INTERFACE iMover

METHOD ActivateTrack : BOOL
VAR_INPUT
	Track	: REFERENCE TO Track;
END_VAR
END_METHOD

{attribute 'monitoring' := 'call'}
PROPERTY CurrentDestinationPosition : LREAL
GET
END_GET
END_PROPERTY

{attribute 'monitoring' := 'call'}
PROPERTY CurrentMoveType : MoverCommandType_enum
GET
END_GET
END_PROPERTY

PROPERTY CurrentObjective : String
GET
END_GET
END_PROPERTY

PROPERTY CurrentTrack : POINTER TO Track
GET
END_GET
END_PROPERTY

METHOD Cyclic : iMover
VAR_IN_OUT
	GroupReference		: AXES_GROUP_REF;
END_VAR
END_METHOD

METHOD CyclicTrack : BOOL
VAR
END_VAR
END_METHOD

METHOD Disable : iMover
VAR_INPUT
END_VAR
END_METHOD

METHOD Enable : iMover
VAR_INPUT
END_VAR
END_METHOD

METHOD GroupStop : iMover
VAR_INPUT
END_VAR
END_METHOD

METHOD Halt : iMover
VAR_INPUT
END_VAR
END_METHOD

PROPERTY IsTrackReady : BOOL
GET
END_GET
END_PROPERTY

METHOD LogUserEvent : iMover
VAR_INPUT
	String1	: STRING;	// First content section of user-event message
	String2 : STRING;	// Second content section of user-event message
	String3 : STRING;	// Third content section of user-event message
END_VAR
END_METHOD

METHOD PUBLIC MoveToPosition : iMover
VAR_INPUT
	
	DestinationPosition		: LREAL;	// position on track for a shuttle to move towards

END_VAR
END_METHOD

METHOD MoveToStation : iMover
VAR_INPUT
	DestinationStation	: REFERENCE TO Station;	
END_VAR
END_METHOD

METHOD MoveVelocity : iMover
VAR_INPUT
	DesiredVelocity : LREAL;		//The velocity to be commanded [mm/s]
END_VAR
END_METHOD

PROPERTY Payload : Payload_TYP
GET
END_GET
SET
END_SET
END_PROPERTY

METHOD ReissueCommand : iMover
VAR_INPUT
END_VAR
END_METHOD


METHOD SetAcceleration : iMover
VAR_INPUT
	Acceleration	: LREAL;
END_VAR
END_METHOD

METHOD SetDeceleration : iMover
VAR_INPUT
	Deceleration	: LREAL;
END_VAR
END_METHOD

METHOD SetDirection : iMover
VAR_INPUT
	Direction		: Tc3_Mc3Definitions.MC_Direction;
END_VAR
END_METHOD

METHOD SetJerk : iMover
VAR_INPUT
	Jerk		: LREAL;
END_VAR
END_METHOD

METHOD SetVelocity : iMover
VAR_INPUT
	Velocity		: LREAL;		// Updates Mover's internal velocity parameter. Takes effect immediately. [mm/s]
END_VAR
END_METHOD

METHOD SyncToAxis : iMover
VAR_INPUT
	
	MasterAxis		: REFERENCE TO AXIS_REF;
	MasterSyncPos	: LREAL;	// Master sync position (nonmodulo), where the input axis will be located when first synchronized
	SlaveSyncPos	: LREAL;	// Mover sync position, where the mover will be located when first synchronized
	SyncStrategy	: MC_SYNC_STRATEGY;	// Direction input
	
END_VAR
END_METHOD

METHOD SyncToMover : iMover
VAR_INPUT

	MasterMover		: REFERENCE TO Mover;	// Synchronization master mover, whose position to follow. Further motion commands break the pairing
	Gap				: LREAL;				// Gap distance to lead mover. Positive values indicate following, negative values indicate leading

END_VAR
END_METHOD

END_INTERFACE

(* stored: Version 1.1.0.1, ProductVersion 3.1.4024.12
   Itf iMover: Id {30ffe45f-c01a-49ae-9d19-23395eddd7e8}
   Folder Methods: Id {1b23c83c-1258-4c4f-a9ad-a029b20875d0}
   Folder Properties: Id {73a4fa43-0d07-4dea-a761-2d7dc373ee4f}
   Method ActivateTrack: Id {0340ebdc-9de8-0f0c-175a-ccd19ec99ec0}
   Property CurrentDestinationPosition: Id {fd336655-1b12-4c85-8800-888e616a0190}
   Get Get: Id {3855cb66-22eb-461a-b098-b3ca2fe0f4f3}
   Property CurrentMoveType: Id {f31956ff-9981-42ba-a963-53182be5a6a1}
   Get Get: Id {4f4d6df0-727b-4d83-aa6a-31cf10efdd21}
   Property CurrentObjective: Id {8ebf7eff-2b0b-45f9-8604-dc48a6c2dec6}
   Get Get: Id {1c8cee4d-d0d3-4396-aef2-3ace7cdfef3e}
   Property CurrentTrack: Id {6df508fb-5bd5-0e4f-32b6-ad8f8b706833}
   Get Get: Id {a9690824-dbea-0ac9-0859-6bf4b97c3449}
   Method Cyclic: Id {b891277c-4d72-4aed-a650-47e395d59c1f}
   Method CyclicTrack: Id {3e3500dc-85cc-0f0e-23f9-0a487fad9df8}
   Method Disable: Id {d596b2ea-b33b-4163-8d7c-887245d1fbda}
   Method Enable: Id {9670332c-ffbe-4d1e-8081-d250b5368f10}
   Method GroupStop: Id {3415d362-731d-4eed-aa29-ec6fe9ada72d}
   Method Halt: Id {75fb2e90-af06-4361-8343-b02ee21a7773}
   Property IsTrackReady: Id {a749704e-a727-05fa-1be8-d11fd5732682}
   Get Get: Id {3d58532e-56d6-0a5a-0811-67af41cc16bc}
   Method LogUserEvent: Id {24391ec1-ea2c-453c-9dee-5da9dcff0b7b}
   Method MoveToPosition: Id {12a28052-bce3-440a-bab1-51b28f359a72}
   Method MoveToStation: Id {1d1440c0-f172-4e49-adaf-b20085e83a8c}
   Method MoveVelocity: Id {86b32a6f-8247-4d7d-b5bb-30abae20d537}
   Property Payload: Id {8debfc3a-ede6-452a-8f81-b4825ce39b3b}
   Get Get: Id {80534c46-bb57-4e05-bca0-e1e88d880aac}
   Set Set: Id {f79463b1-b92f-424b-a739-aa6b1256efa9}
   Method ReissueCommand: Id {1fc1edba-27e0-4034-90b8-62d930acd5b9}
   Method SetAcceleration: Id {8d0e79e2-9192-4e14-ba95-b7dae3613c61}
   Method SetDeceleration: Id {04f2ddea-3c35-4990-b2b0-631376080d3c}
   Method SetDirection: Id {af950f72-a593-4951-9d27-c94a586f0a6a}
   Method SetJerk: Id {7c744f28-4b51-4d53-bcdc-6b5a1cdf2938}
   Method SetVelocity: Id {335b28ab-3de7-4b93-9e44-7bd94a4041e5}
   Method SyncToAxis: Id {5a310de1-52da-0514-1130-76a03f36818d}
   Method SyncToMover: Id {818e2706-7bf4-42d7-a370-2480751106b6} *)
